TYPE ST_OperationVars_Genset :
STRUCT 
	b_manualStart			: BOOL;
END_STRUCT
END_TYPE

(* stored: Version 1.1.0.1, ProductVersion 3.1.4026.18
   DUT ST_OperationVars_Genset: Id {2e99b50b-23cd-4fb8-9862-69c96b0eaf2b} *)
